TYPE ST_Custom_HMI EXTENDS ST_HmiFunction :
	STRUCT
	END_STRUCT
END_TYPE

(* stored: Version 1.1.0.1, ProductVersion 3.1.4026.18
   DUT ST_Custom_HMI: Id {6e4e836e-01d9-49d9-878f-9512c4c65e71} *)
